Fanuc KAREL source: NC0079.KL

-- PROVISIONAL review KL for V940-1; original PC SHA256 5c408d0967d51876e9b807fad97f49f91a6d489cdcb2891a9f015536bcfea2a3
-- Incomplete behavior may be omitted. Consult companion uncertainty JSON. Do not deploy.
PROGRAM NC0079
%NOLOCKGROUP
-- UNRESOLVED_LOCAL_POOL 1 cells at code offset 3; source declarations unknown
-- DIRECT_LOCAL_WORD_ACCESS alone does not prove INTEGER, REAL, or BOOLEAN
BEGIN
  -- V9_OWNER_INTERVAL_HINT [6,116),[11,114),[16,112),[21,110),[26,108),[31,106),[36,104),[41,102),[46,100),[51,98),[56,96),[61,94),[66,92),[71,90),[76,88); structural only; source/VM held
  -- V9_EXPOSED_INDEXED_TABLE_HINT layout=0001; 30 counted words exposed once; source arms/runtime held
  -- UNRESOLVED_PC offsets 0-8; opcodes 2B,2C,7B
  -- UNRESOLVED_PC offsets 13-20; opcodes 9D,23
  -- UNRESOLVED_PC offsets 25-42; opcodes 21,2E,59,79
  -- UNRESOLVED_PC offsets 47-64; opcodes 21,2E,59,79
  -- UNRESOLVED_PC offsets 69-86; opcodes 21,2E,59,79
  -- UNRESOLVED_PC offsets 91-108; opcodes 21,2E,59,79
  -- UNRESOLVED_PC offsets 113-130; opcodes 21,2E,59,79
  -- UNRESOLVED_PC offsets 135-152; opcodes 21,2E,59,79
  -- UNRESOLVED_PC offsets 157-174; opcodes 21,2E,59,79
  -- UNRESOLVED_PC offsets 179-196; opcodes 21,2E,59,79
  -- UNRESOLVED_PC offsets 201-218; opcodes 21,2E,59,79
  -- UNRESOLVED_PC offsets 223-240; opcodes 21,2E,59,79
  -- UNRESOLVED_PC offsets 245-262; opcodes 21,2E,59,79
  -- UNRESOLVED_PC offsets 267-284; opcodes 21,2E,59,79
  -- UNRESOLVED_PC offsets 289-306; opcodes 21,2E,59,79
  -- UNRESOLVED_PC offsets 311-328; opcodes 21,2E,59,79
  -- UNRESOLVED_PC offsets 333-350; opcodes 21,2E,59,79
  -- UNRESOLVED_PC offsets 355-369; opcodes 21,9D,52,23
  -- UNRESOLVED_PC offsets 374-379; opcodes 7A
  -- UNRESOLVED_PC offsets 384-389; opcodes 7A
  -- UNRESOLVED_PC offsets 394-399; opcodes 7A
  -- UNRESOLVED_PC offsets 404-409; opcodes 7A
  -- UNRESOLVED_PC offsets 414-419; opcodes 7A
  -- UNRESOLVED_PC offsets 424-429; opcodes 7A
  -- UNRESOLVED_PC offsets 434-439; opcodes 7A
  -- UNRESOLVED_PC offsets 444-449; opcodes 7A
  -- UNRESOLVED_PC offsets 454-459; opcodes 7A
  -- UNRESOLVED_PC offsets 464-469; opcodes 7A
  -- UNRESOLVED_PC offsets 474-479; opcodes 7A
  -- UNRESOLVED_PC offsets 484-489; opcodes 7A
  -- UNRESOLVED_PC offsets 494-499; opcodes 7A
  -- UNRESOLVED_PC offsets 504-509; opcodes 7A
  -- UNRESOLVED_PC offsets 514-519; opcodes 7A
  -- UNRESOLVED_PC offsets 524-528; opcodes 7F
  -- UNRESOLVED_PC offsets 533-537; opcodes 27,AA
  -- UNRESOLVED_PC offsets 542-546; opcodes 7F
END NC0079
